// TIA Portal V18 export
// export: Created 2025-12-01T12:38:01.0658705Z, ExportSetting None, DisplayName Totally Integrated Automation Portal, DisplayVersion V18 Update 5, DisplayName TIA Portal Openness, DisplayVersion V18 Update 5, DisplayName TIA Portal Teamcenter Gateway, DisplayVersion V18, DisplayName TIA Portal Version Control Interface, DisplayVersion V18, DisplayName STEP 7 Professional, DisplayVersion V18 Update 5, DisplayName STEP 7 Safety, DisplayVersion V18, DisplayName WinCC Professional, DisplayVersion V18 Update 5
FUNCTION_BLOCK "FB_Stopper"   // FB4001, LAD
{ S7_Optimized_Access := 'FALSE' }
// stored: AutoNumber false, SetENOAutomatically false
   VAR_INPUT
      iSysInface : "RCS_SysComInterface_V1";
      iSensor : Bool;   // 本站托盘到位
      iNextSensor : Bool;   // 后站托盘到位
      iNextValve : Bool;   // 后站挡停输出
      iPresentDwell : Time := T#0.3s;   // 本站到位传感器延时
      iNextEmptyDwell : Time := T#10s;   // 后站托盘到位传感器延时
      iReleaseClear : Bool;   // 托盘释放允许
      iReleaseDwell : Time := T#1s;   // 托盘已流出延时
      iReleaseFaultTimer : Time := T#1s;   // 托盘流出超时延时
      iReachFaultTimer : Time := T#5s;   // 托盘流入后站超时延时
   END_VAR
   VAR_OUTPUT
      oValve : Bool;   // 本站挡停输出
      oReleaseCompleted : Bool;   // 释放完成
      oReleaseFault : Bool;   // 托盘流走超时
      oReachFault : Bool;   // 后站托盘接收超时
      oNotClear : Bool;   // 手动释放中
   END_VAR
   VAR_IN_OUT
      io_Dev : "ST_Stopper";
   END_VAR
   VAR
      Stopper : Struct
         Sensor : Bool;
         Valve : Bool;
         NextSensor : Bool;
         NextValve : Bool;
         NextFullSensor : Bool;
         PresentDwell : TON_TIME;
         NextEmptyDwell : TON_TIME;
         NextFullDwell : TON_TIME;
         ReleaseClear : Bool;
         ReleaseMemory : Bool;
         ReleaseDwell : TON_TIME;
         ReleasePB : Bool;
         NotClear : Bool;
         NextEmptyMemory : Bool;
         ReleaseCompleted : Bool;
         ReleaseFaultTimer : TON_TIME;
         ReachFaultTimer : TON_TIME;
      END_STRUCT;
   END_VAR
BEGIN

REGION Network 1: 输入输出映射 / Input output map
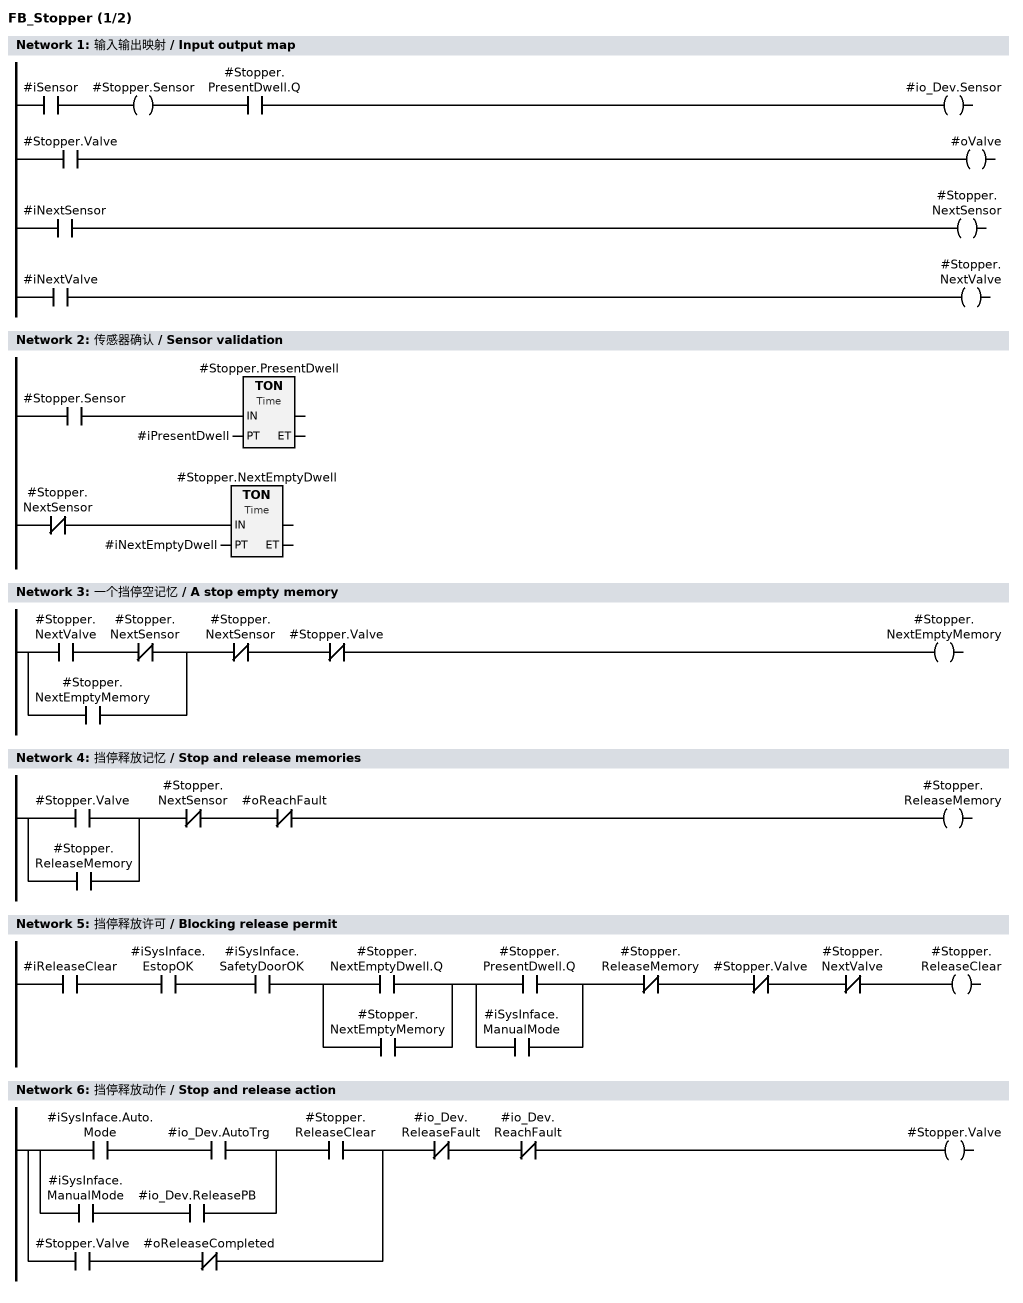
   RUNG wire#powerrail
      Contact( #iSensor )
      Coil( #Stopper.Sensor )
      Contact( #Stopper.PresentDwell.Q )
      Coil( #io_Dev.Sensor )
   END_RUNG
   RUNG wire#powerrail
      Contact( #Stopper.Valve )
      Coil( #oValve )
   END_RUNG
   RUNG wire#powerrail
      Contact( #iNextSensor )
      Coil( #Stopper.NextSensor )
   END_RUNG
   RUNG wire#powerrail
      Contact( #iNextValve )
      Coil( #Stopper.NextValve )
   END_RUNG
   // the same network as SCL:
   #Stopper.Sensor := #iSensor;
   #io_Dev.Sensor := #iSensor AND #Stopper.PresentDwell.Q;
   #oValve := #Stopper.Valve;
   #Stopper.NextSensor := #iNextSensor;
   #Stopper.NextValve := #iNextValve;
END_REGION

REGION Network 2: 传感器确认 / Sensor validation
   RUNG wire#powerrail
      Contact( #Stopper.Sensor )
      { S7_Templates := "time_type := Time" } #Stopper.PresentDwell.TON(pt := #iPresentDwell, et =>)
   END_RUNG
   RUNG wire#powerrail
      I_Contact( #Stopper.NextSensor )
      { S7_Templates := "time_type := Time" } #Stopper.NextEmptyDwell.TON(pt := #iNextEmptyDwell, et =>)
   END_RUNG
   // the same network as SCL:
   #Stopper.PresentDwell.TON(IN := #Stopper.Sensor, PT := #iPresentDwell);
   #Stopper.NextEmptyDwell.TON(IN := NOT #Stopper.NextSensor, PT := #iNextEmptyDwell);
END_REGION

REGION Network 3: 一个挡停空记忆 / A stop empty memory
   RUNG wire#powerrail
      Contact( #Stopper.NextValve )
      I_Contact( #Stopper.NextSensor )
      wire#w1
      I_Contact( #Stopper.NextSensor )
      I_Contact( #Stopper.Valve )
      Coil( #Stopper.NextEmptyMemory )
   END_RUNG
   RUNG wire#powerrail
      Contact( #Stopper.NextEmptyMemory )
   END_RUNG wire#w1
   // the same network as SCL:
   #Stopper.NextEmptyMemory := ((#Stopper.NextValve AND NOT #Stopper.NextSensor) OR #Stopper.NextEmptyMemory) AND NOT #Stopper.NextSensor AND NOT #Stopper.Valve;
END_REGION

REGION Network 4: 挡停释放记忆 / Stop and release memories
   RUNG wire#powerrail
      Contact( #Stopper.Valve )
      wire#w1
      I_Contact( #Stopper.NextSensor )
      I_Contact( #oReachFault )
      Coil( #Stopper.ReleaseMemory )
   END_RUNG
   RUNG wire#powerrail
      Contact( #Stopper.ReleaseMemory )
   END_RUNG wire#w1
   // the same network as SCL:
   #Stopper.ReleaseMemory := (#Stopper.Valve OR #Stopper.ReleaseMemory) AND NOT #Stopper.NextSensor AND NOT #oReachFault;
END_REGION

REGION Network 5: 挡停释放许可 / Blocking release permit
   RUNG wire#powerrail
      Contact( #iReleaseClear )
      Contact( #iSysInface.EstopOK )
      Contact( #iSysInface.SafetyDoorOK )
      wire#w1
      Contact( #Stopper.NextEmptyDwell.Q )
      wire#w2
      Contact( #Stopper.PresentDwell.Q )
      wire#w3
      I_Contact( #Stopper.ReleaseMemory )
      I_Contact( #Stopper.Valve )
      I_Contact( #Stopper.NextValve )
      Coil( #Stopper.ReleaseClear )
   END_RUNG
   RUNG wire#w1
      Contact( #Stopper.NextEmptyMemory )
   END_RUNG wire#w2
   RUNG wire#w2
      Contact( #iSysInface.ManualMode )
   END_RUNG wire#w3
   // the same network as SCL:
   #Stopper.ReleaseClear := #iReleaseClear AND #iSysInface.EstopOK AND #iSysInface.SafetyDoorOK AND (#Stopper.NextEmptyDwell.Q OR #Stopper.NextEmptyMemory) AND (#Stopper.PresentDwell.Q OR #iSysInface.ManualMode) AND NOT #Stopper.ReleaseMemory AND NOT #Stopper.Valve AND NOT #Stopper.NextValve;
END_REGION

REGION Network 6: 挡停释放动作 / Stop and release action
   RUNG wire#powerrail
      Contact( #iSysInface.Auto.Mode )
      Contact( #io_Dev.AutoTrg )
      wire#w1
      Contact( #Stopper.ReleaseClear )
      wire#w2
      I_Contact( #io_Dev.ReleaseFault )
      I_Contact( #io_Dev.ReachFault )
      Coil( #Stopper.Valve )
   END_RUNG
   RUNG wire#powerrail
      Contact( #iSysInface.ManualMode )
      Contact( #io_Dev.ReleasePB )
   END_RUNG wire#w1
   RUNG wire#powerrail
      Contact( #Stopper.Valve )
      I_Contact( #oReleaseCompleted )
   END_RUNG wire#w2
   // the same network as SCL:
   #Stopper.Valve := ((((#iSysInface.Auto.Mode AND #io_Dev.AutoTrg) OR (#iSysInface.ManualMode AND #io_Dev.ReleasePB)) AND #Stopper.ReleaseClear) OR (#Stopper.Valve AND NOT #oReleaseCompleted)) AND NOT #io_Dev.ReleaseFault AND NOT #io_Dev.ReachFault;
END_REGION

REGION Network 7: 释放完成信号 / Release completion signal
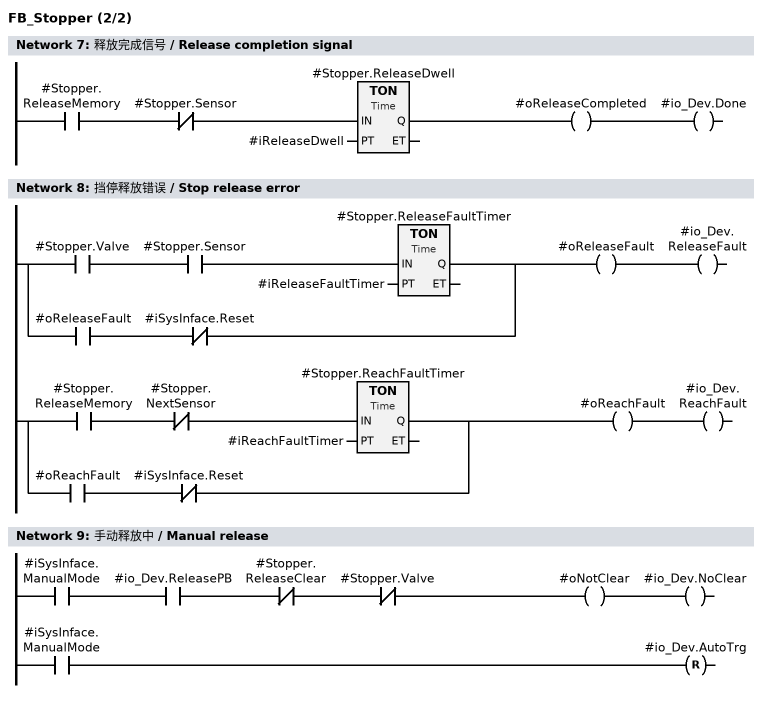
   RUNG wire#powerrail
      Contact( #Stopper.ReleaseMemory )
      I_Contact( #Stopper.Sensor )
      { S7_Templates := "time_type := Time" } #Stopper.ReleaseDwell.TON(pt := #iReleaseDwell, et =>)
      Coil( #oReleaseCompleted )
      Coil( #io_Dev.Done )
   END_RUNG
   // the same network as SCL:
   #Stopper.ReleaseDwell.TON(IN := #Stopper.ReleaseMemory AND NOT #Stopper.Sensor, PT := #iReleaseDwell);
   #oReleaseCompleted := #Stopper.ReleaseDwell.Q;
   #io_Dev.Done := #Stopper.ReleaseDwell.Q;
END_REGION

REGION Network 8: 挡停释放错误 / Stop release error
   RUNG wire#powerrail
      Contact( #Stopper.Valve )
      Contact( #Stopper.Sensor )
      { S7_Templates := "time_type := Time" } #Stopper.ReleaseFaultTimer.TON(pt := #iReleaseFaultTimer, et =>)
      wire#w1
      Coil( #oReleaseFault )
      Coil( #io_Dev.ReleaseFault )
   END_RUNG
   RUNG wire#powerrail
      Contact( #oReleaseFault )
      I_Contact( #iSysInface.Reset )
   END_RUNG wire#w1
   RUNG wire#powerrail
      Contact( #Stopper.ReleaseMemory )
      I_Contact( #Stopper.NextSensor )
      { S7_Templates := "time_type := Time" } #Stopper.ReachFaultTimer.TON(pt := #iReachFaultTimer, et =>)
      wire#w2
      Coil( #oReachFault )
      Coil( #io_Dev.ReachFault )
   END_RUNG
   RUNG wire#powerrail
      Contact( #oReachFault )
      I_Contact( #iSysInface.Reset )
   END_RUNG wire#w2
   // the same network as SCL:
   #Stopper.ReleaseFaultTimer.TON(IN := #Stopper.Valve AND #Stopper.Sensor, PT := #iReleaseFaultTimer);
   #oReleaseFault := #Stopper.ReleaseFaultTimer.Q OR (#oReleaseFault AND NOT #iSysInface.Reset);
   #io_Dev.ReleaseFault := #oReleaseFault;
   #Stopper.ReachFaultTimer.TON(IN := #Stopper.ReleaseMemory AND NOT #Stopper.NextSensor,
                           PT := #iReachFaultTimer);
   #oReachFault := #Stopper.ReachFaultTimer.Q OR (#oReachFault AND NOT #iSysInface.Reset);
   #io_Dev.ReachFault := #oReachFault;
END_REGION

REGION Network 9: 手动释放中 / Manual release
   RUNG wire#powerrail
      Contact( #iSysInface.ManualMode )
      Contact( #io_Dev.ReleasePB )
      I_Contact( #Stopper.ReleaseClear )
      I_Contact( #Stopper.Valve )
      Coil( #oNotClear )
      Coil( #io_Dev.NoClear )
   END_RUNG
   RUNG wire#powerrail
      Contact( #iSysInface.ManualMode )
      R_Coil( #io_Dev.AutoTrg )
   END_RUNG
   // the same network as SCL:
   #oNotClear := #iSysInface.ManualMode AND #io_Dev.ReleasePB AND NOT #Stopper.ReleaseClear AND NOT #Stopper.Valve;
   #io_Dev.NoClear := #oNotClear;
   IF #iSysInface.ManualMode THEN #io_Dev.AutoTrg := FALSE; END_IF;
END_REGION
END_FUNCTION_BLOCK
